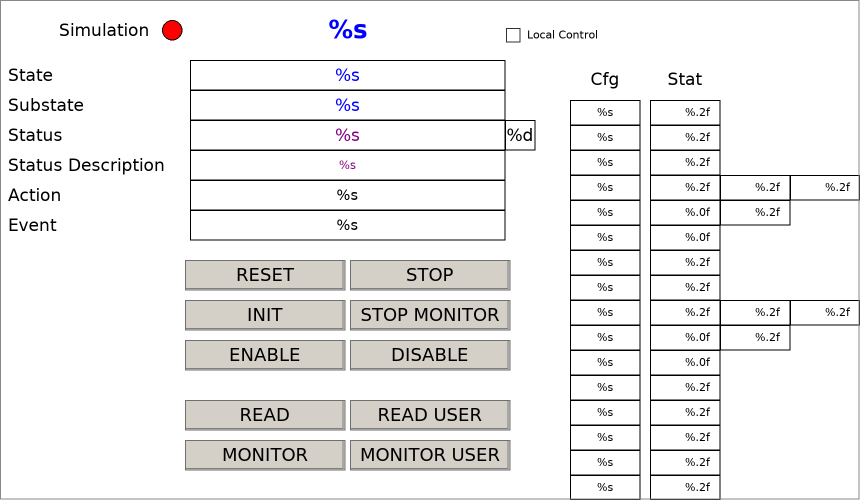
VISUALIZATION GUI_TEMPLATE_LAKESHORE_TCP_RT_336  // 860x500
VAR_IN_OUT
	m_Instance:	FB_LAKESHORE_TCP_RT;
END_VAR
    Rectangle (190,60 315x30), "%s", text variable: m_Instance.stat.sState
    Rectangle (190,90 315x30), "%s", text variable: m_Instance.stat.sSubstate
    Button (185,260 160x30), "RESET", input disabled if: (m_Instance.stat.bLocal = FALSE) <> 0
        OnMouseClick: execute { m_Instance.ctrl.nCommand := E_RS_COMMAND.RESET; m_Instance.ctrl.bExecute := TRUE; }
    Button (185,300 160x30), "INIT", input disabled if: (m_Instance.stat.bLocal = FALSE) <> 0
        OnMouseClick: execute { m_Instance.ctrl.nCommand := E_RS_COMMAND.INIT; m_Instance.ctrl.bExecute := TRUE; }
    Button (350,260 160x30), "STOP", input disabled if: (m_Instance.stat.bLocal = FALSE) <> 0
        OnMouseClick: execute { m_Instance.ctrl.nCommand := E_RS_COMMAND.STOP; m_Instance.ctrl.bExecute := TRUE; }
    Button (185,340 160x30), "ENABLE", input disabled if: (m_Instance.stat.bLocal = FALSE) <> 0
        OnMouseClick: execute { m_Instance.ctrl.nCommand := E_RS_COMMAND.ENABLE; m_Instance.ctrl.bExecute := TRUE; }
    Button (350,340 160x30), "DISABLE", input disabled if: (m_Instance.stat.bLocal = FALSE) <> 0
        OnMouseClick: execute { m_Instance.ctrl.nCommand := E_RS_COMMAND.DISABLE; m_Instance.ctrl.bExecute := TRUE; }
    Rectangle (5,60 180x30), "State"
    Rectangle (5,90 180x30), "Substate"
    Rectangle (190,120 315x30), "%s", text variable: m_Instance.stat.sStatus
    Rectangle (190,150 315x30), "%s", text variable: m_Instance.stat.sErrorText
    Rectangle (5,120 180x30), "Status"
    Rectangle (5,150 180x30), "Status Description"
    Rectangle (190,180 315x30), "%s", text variable: m_Instance.stat.sActionDesc
    Rectangle (190,210 315x30), "%s", text variable: m_Instance.stat.sEventDesc
    Rectangle (5,180 180x30), "Action"
    Rectangle (5,210 180x30), "Event"
    Rectangle (232,12 232x35), "%s", text variable: m_Instance.in_sName
    Rectangle (574,64 62x30), "Cfg"
    Checkbox (504,20 116x30), "Local Control", variable: m_Instance.stat.bLocal
    Rectangle (505,120 30x30), "%d", text variable: m_Instance.stat.nStatus
    Button (185,400 160x30), "READ", tooltip "Single read of all commands in the configuration", input disabled if: (m_Instance.stat.bLocal = FALSE) <> 0
        OnMouseClick: execute { m_Instance.ctrl.nCommand := E_RS_COMMAND.READ; m_Instance.ctrl.bExecute := TRUE; }
    Button (350,400 160x30), "READ USER", tooltip "Single read of user command", input disabled if: (m_Instance.stat.bLocal = FALSE) <> 0
        OnMouseClick: execute { m_Instance.ctrl.nCommand := E_RS_COMMAND.READ_USER; m_Instance.ctrl.bExecute := TRUE; }
    Button (185,440 160x30), "MONITOR", tooltip "Continuously read all commands in the configuration", input disabled if: (m_Instance.stat.bLocal = FALSE) <> 0
        OnMouseClick: execute { m_Instance.ctrl.nCommand := E_RS_COMMAND.MONITOR; m_Instance.ctrl.bExecute := TRUE; }
    Button (350,440 160x30), "MONITOR USER", tooltip "Continuously read the User command", input disabled if: (m_Instance.stat.bLocal = FALSE) <> 0
        OnMouseClick: execute { m_Instance.ctrl.nCommand := E_RS_COMMAND.MONITOR_USER; m_Instance.ctrl.bExecute := TRUE; }
    Rectangle (570,100 70x25), "%s", text variable: m_Instance.cfg.cmdList_Read[1].cmd
    Rectangle (570,125 70x25), "%s", text variable: m_Instance.cfg.cmdList_Read[2].cmd
    Rectangle (570,150 70x25), "%s", text variable: m_Instance.cfg.cmdList_Read[3].cmd
    Rectangle (570,175 70x25), "%s", text variable: m_Instance.cfg.cmdList_Read[4].cmd
    Rectangle (570,200 70x25), "%s", text variable: m_Instance.cfg.cmdList_Read[5].cmd
    Rectangle (570,225 70x25), "%s", text variable: m_Instance.cfg.cmdList_Read[6].cmd
    Rectangle (570,250 70x25), "%s", text variable: m_Instance.cfg.cmdList_Read[7].cmd
    Rectangle (570,275 70x25), "%s", text variable: m_Instance.cfg.cmdList_Read[8].cmd
    Rectangle (570,300 70x25), "%s", text variable: m_Instance.cfg.cmdList_Read[9].cmd
    Rectangle (570,325 70x25), "%s", text variable: m_Instance.cfg.cmdList_Read[10].cmd
    Rectangle (570,350 70x25), "%s", text variable: m_Instance.cfg.cmdList_Read[11].cmd
    Rectangle (570,375 70x25), "%s", text variable: m_Instance.cfg.cmdList_Read[12].cmd
    Rectangle (570,400 70x25), "%s", text variable: m_Instance.cfg.cmdList_Read[13].cmd
    Rectangle (570,425 70x25), "%s", text variable: m_Instance.cfg.cmdList_Read[14].cmd
    Rectangle (570,450 70x25), "%s", text variable: m_Instance.cfg.cmdList_Read[15].cmd
    Rectangle (570,475 70x25), "%s", text variable: m_Instance.cfg.cmdList_Read[16].cmd
    Rectangle (650,100 70x25), "%.2f", text variable: m_Instance.stat.lrArrReadings[0].lrValue
    Rectangle (650,125 70x25), "%.2f", text variable: m_Instance.stat.lrArrReadings[1].lrValue
    Rectangle (650,150 70x25), "%.2f", text variable: m_Instance.stat.lrArrReadings[2].lrValue
    Rectangle (650,175 70x25), "%.2f", text variable: m_Instance.stat.lrArrReadings[3].lrValue
    Rectangle (720,175 70x25), "%.2f", text variable: m_Instance.stat.lrArrReadings[4].lrValue
    Rectangle (790,175 70x25), "%.2f", text variable: m_Instance.stat.lrArrReadings[5].lrValue
    Rectangle (650,200 70x25), "%.0f", text variable: m_Instance.stat.lrArrReadings[6].lrValue
    Rectangle (650,225 70x25), "%.0f", text variable: m_Instance.stat.lrArrReadings[8].lrValue
    Rectangle (650,250 70x25), "%.2f", text variable: m_Instance.stat.lrArrReadings[9].lrValue
    Rectangle (650,275 70x25), "%.2f", text variable: m_Instance.stat.lrArrReadings[10].lrValue
    Rectangle (720,300 70x25), "%.2f", text variable: m_Instance.stat.lrArrReadings[12].lrValue
    Rectangle (790,300 70x25), "%.2f", text variable: m_Instance.stat.lrArrReadings[13].lrValue
    Rectangle (650,300 70x25), "%.2f", text variable: m_Instance.stat.lrArrReadings[11].lrValue
    Rectangle (720,325 70x25), "%.2f", text variable: m_Instance.stat.lrArrReadings[15].lrValue
    Rectangle (650,350 70x25), "%.0f", text variable: m_Instance.stat.lrArrReadings[16].lrValue
    Rectangle (650,375 70x25), "%.2f", text variable: m_Instance.stat.lrArrReadings[17].lrValue
    Rectangle (650,400 70x25), "%.2f", text variable: m_Instance.stat.lrArrReadings[18].lrValue
    Rectangle (650,425 70x25), "%.2f", text variable: m_Instance.stat.lrArrReadings[19].lrValue
    Rectangle (650,450 70x25), "%.2f", text variable: m_Instance.stat.lrArrReadings[20].lrValue
    Rectangle (650,475 70x25), "%.2f", text variable: m_Instance.stat.lrArrReadings[21].lrValue
    Rectangle (654,64 62x30), "Stat"
    Button (350,300 160x30), "STOP MONITOR", tooltip "Stop Monitoring if in OP/MONITORIN state.", input disabled if: (m_Instance.stat.bLocal = FALSE) <> 0
        OnMouseClick: execute { m_Instance.ctrl.nCommand := E_RS_COMMAND.STOPMON; m_Instance.ctrl.bExecute := TRUE; }
    Rectangle (56,15 101x30), "Simulation", invisible if: (m_Instance.stat.bSimulation=FALSE)
    Ellipse (162,20 20x20), tooltip "GREEN=Initialized RED=Not-initialized", text variable: m_Instance.stat.bInitialised, invisible if: (m_Instance.stat.bSimulation=FALSE)
    Rectangle (720,200 70x25), "%.2f", text variable: m_Instance.stat.lrArrReadings[7].lrValue
    Rectangle (650,325 70x25), "%.0f", text variable: m_Instance.stat.lrArrReadings[14].lrValue
END_VISUALIZATION

(* stored: Version 1.1.0.1, ProductVersion 3.1.4024.9
   Visu GUI_TEMPLATE_LAKESHORE_TCP_RT_336: Id {b5f252a8-2d21-4e05-bf3a-1657825f8094} *)
